// Mitsubishi GX Developer project: 6.0丝杠4圈（单感应柱改诊断模式改延时方式）--4-6T通用20231021   PLC: FX2N

PROGRAM MAIN
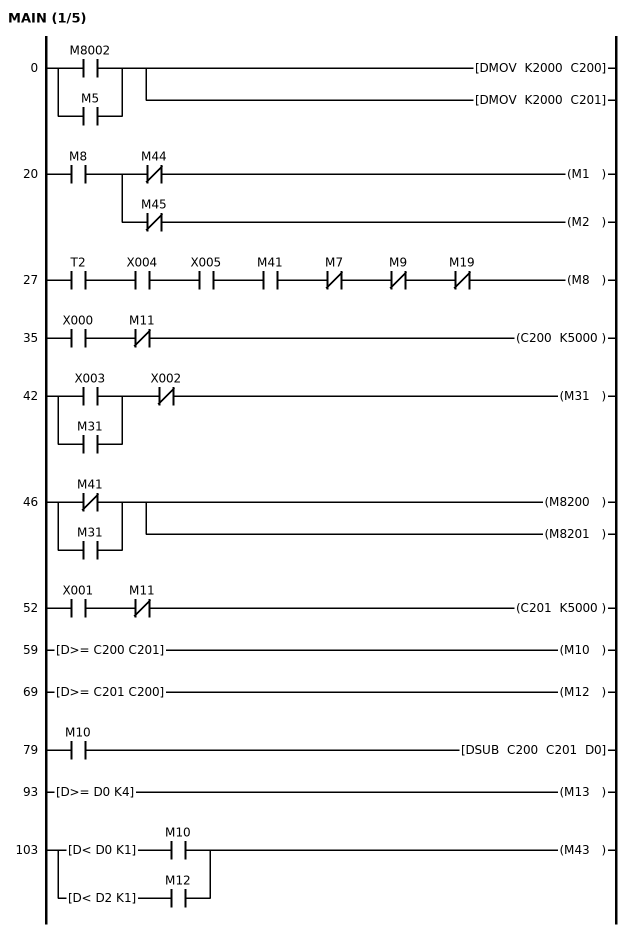
0     LD      M8002
      OR      M5
      DMOV    K2000 C200
        [note] 初始化
      DMOV    K2000 C201
20    LD      M8
      MPS
      ANI     M44
      OUT     M1
        [note] 上升程序段    上升驱动段
      MPP
      ANI     M45
      OUT     M2
27    LD      T2
      AND     X004
      AND     X005
      AND     M41
      ANI     M7
      ANI     M9
      ANI     M19
      OUT     M8
35    LD      X000
      ANI     M11
      OUT     C200 K5000
        [note] 计数
42    LD      X003
      OR      M31
      ANI     X002
      OUT     M31
46    LDI     M41
      OR      M31
      OUT     M8200
      OUT     M8201
52    LD      X001
      ANI     M11
      OUT     C201 K5000
59    LDD>=   C200 C201
      OUT     M10
        [note] 数据比较程序段
69    LDD>=   C201 C200
      OUT     M12
79    LD      M10
      DSUB    C200 C201 D0
93    LDD>=   D0 K4
      OUT     M13
103   LDD<    D0 K1
      AND     M10
      LDD<    D2 K1
      AND     M12
      ORB
      OUT     M43
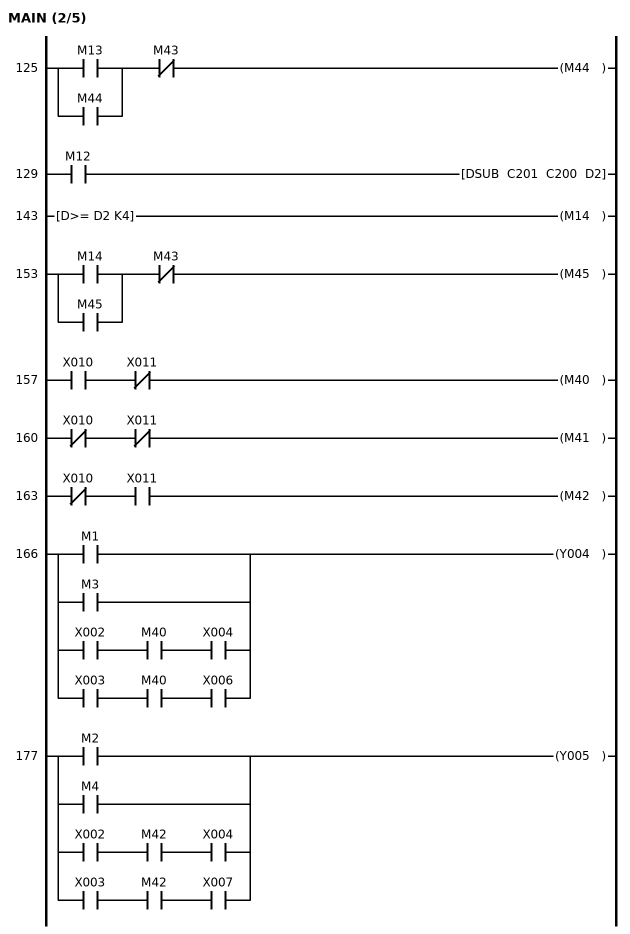
125   LD      M13
      OR      M44
      ANI     M43
      OUT     M44
129   LD      M12
      DSUB    C201 C200 D2
143   LDD>=   D2 K4
      OUT     M14
153   LD      M14
      OR      M45
      ANI     M43
      OUT     M45
157   LD      X010
      ANI     X011
      OUT     M40
160   LDI     X010
      ANI     X011
      OUT     M41
163   LDI     X010
      AND     X011
      OUT     M42
166   LD      M1
      OR      M3
      LD      X002
      AND     M40
      AND     X004
      ORB
      LD      X003
      AND     M40
      AND     X006
      ORB
      OUT     Y004
        [note] 输出端口
177   LD      M2
      OR      M4
      LD      X002
      AND     M42
      AND     X004
      ORB
      LD      X003
      AND     M42
      AND     X007
      ORB
      OUT     Y005
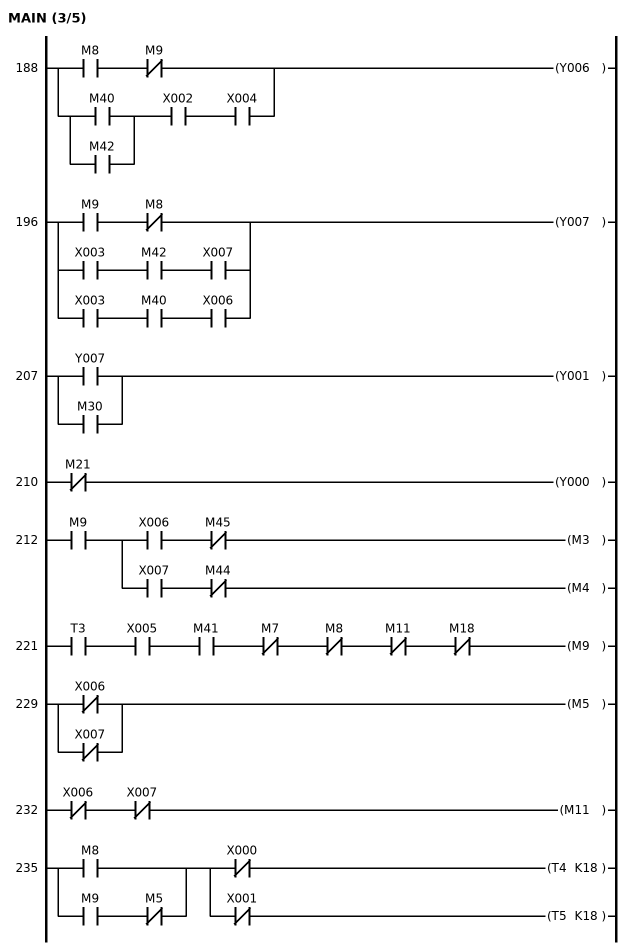
188   LD      M8
      ANI     M9
      LD      M40
      OR      M42
      AND     X002
      AND     X004
      ORB
      OUT     Y006
196   LD      M9
      ANI     M8
      LD      X003
      AND     M42
      AND     X007
      ORB
      LD      X003
      AND     M40
      AND     X006
      ORB
      OUT     Y007
207   LD      Y007
      OR      M30
      OUT     Y001
210   LDI     M21
      OUT     Y000
212   LD      M9
      MPS
      AND     X006
      ANI     M45
      OUT     M3
        [note] 下降程序段
      MPP
      AND     X007
      ANI     M44
      OUT     M4
221   LD      T3
      AND     X005
      AND     M41
      ANI     M7
      ANI     M8
      ANI     M11
      ANI     M18
      OUT     M9
229   LDI     X006
      ORI     X007
      OUT     M5
        [note] 下限清零
232   LDI     X006
      ANI     X007
      OUT     M11
235   LD      M8
      LD      M9
      ANI     M5
      ORB
      MPS
      ANI     X000
      OUT     T4 K18
        [note] 报警程序   霍尔故障
      MPP
      ANI     X001
      OUT     T5 K18
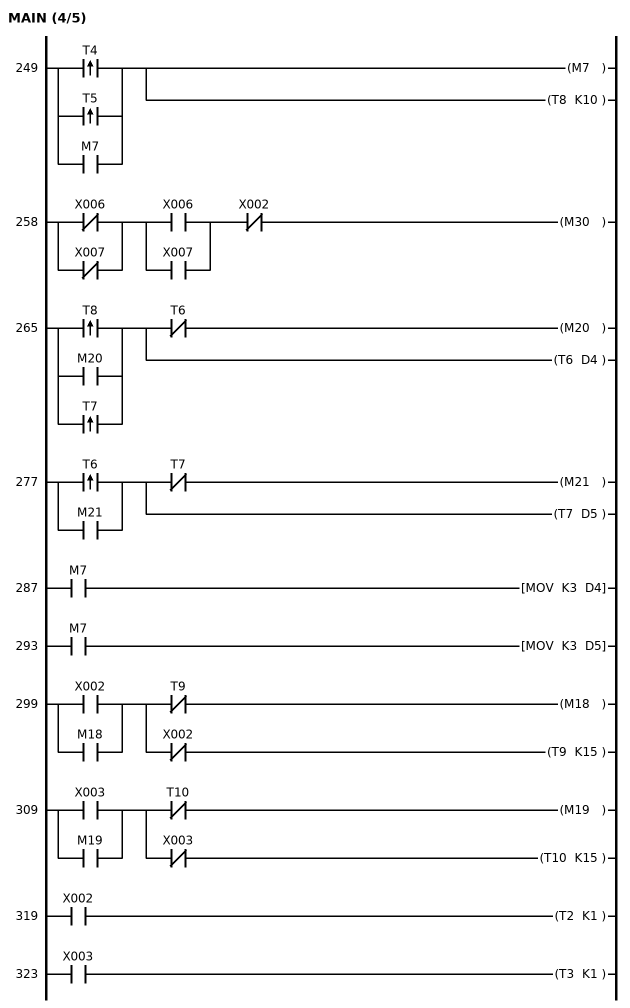
249   LDP     T4
      ORP     T5
      OR      M7
      OUT     M7
      OUT     T8 K10
258   LDI     X006
      ORI     X007
      LD      X006
      OR      X007
      ANB
      ANI     X002
      OUT     M30
        [note] 下限状态
265   LDP     T8
      OR      M20
      ORP     T7
      MPS
      ANI     T6
      OUT     M20
        [note] 双稳态
      MPP
      OUT     T6 D4
277   LDP     T6
      OR      M21
      MPS
      ANI     T7
      OUT     M21
      MPP
      OUT     T7 D5
287   LD      M7
      MOV     K3 D4
        [note] 赋值
293   LD      M7
      MOV     K3 D5
299   LD      X002
      OR      M18
      MPS
      ANI     T9
      OUT     M18
        [note] 上下按键互锁
      MPP
      ANI     X002
      OUT     T9 K15
309   LD      X003
      OR      M19
      MPS
      ANI     T10
      OUT     M19
      MPP
      ANI     X003
      OUT     T10 K15
319   LD      X002
      OUT     T2 K1
323   LD      X003
      OUT     T3 K1
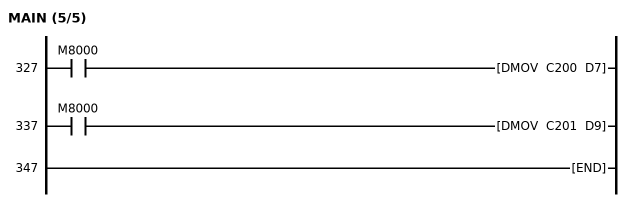
327   LD      M8000
      DMOV    C200 D7
337   LD      M8000
      DMOV    C201 D9
347   END
END_PROGRAM
